FUNCTION_BLOCK ExtControlBehaviour IMPLEMENTS I_Cyclic
VAR
	ThisMover : I_XtsMover;
	LeaveTest: BOOL;
	ArriveTest: BOOL;
	TestMove: BOOL;
	Position: MC_LREAL;
	Velocity: MC_LREAL;
END_VAR

METHOD PUBLIC  Cycle : HRESULT
VAR_INPUT
END_VAR
IF LeaveTest THEN
	ThisMover.TriggerMoverLeave();
END_IF

IF ArriveTest THEN
	ThisMover.TriggerMoverArrive();
END_IF

IF TestMove THEN
	ThisMover.MoveTo(RequiredPosition := Position, MoveVelocity := Velocity, NonModuloMove := FALSE);
	TestMove := FALSE;
END_IF
END_METHOD

PROPERTY MyMover : I_XtsMover
GET
MyMover := ThisMover;
END_GET
SET
ThisMover := MyMover;
END_SET
END_PROPERTY

END_FUNCTION_BLOCK

(* stored: Version 1.1.0.1
   POU ExtControlBehaviour: Id {d3f2ac87-b8f7-4911-b9c2-b9baff5eb1c4}, SpecialFunc None
   Method Cycle: Id {8888b623-da21-4226-add6-1f1bd1a51781}
   Property MyMover: Id {a5c868b0-cac0-4f55-bd66-8ef755b79feb}
   Get Get: Id {587907ca-a173-4213-9ae5-405c4a27d931}
   Set Set: Id {61ecbb90-d62b-4e06-b9a5-e3c58bf4d7f4} *)
